KUKA KRL program: Rack_Azul_Dejar.src, Rack_Azul_Dejar.dat

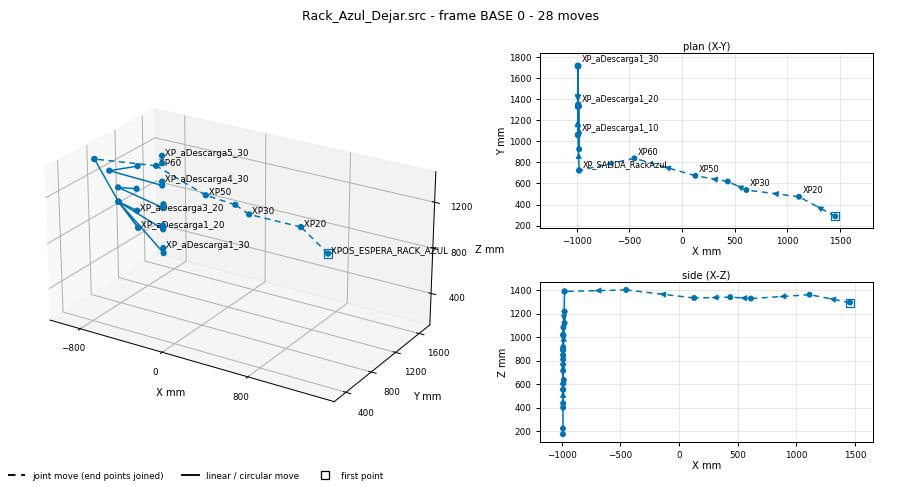
[picture p0: tool path of Rack_Azul_Dejar.src in frame BASE 0, 28 of 41 moves have a stored position in this frame; points joined in program order, loops and branches not executed]
--- Rack_Azul_Dejar.src ---
&ACCESS RVO1
&REL 3149
&COMMENT DEJAR BAT EN RACK AZUL
&PARAM EDITMASK = *
&PARAM TEMPLATE = C:\KRC\Roboter\Template\vorgabe
&PARAM DISKPATH = KRC:\R1\Program\MAFELEC
DEF Rack_Azul_Dejar( )
;FOLD INI;%{PE}
  ;FOLD BASISTECH INI
    GLOBAL INTERRUPT DECL 3 WHEN $STOPMESS==TRUE DO IR_STOPM ( )
    INTERRUPT ON 3
    BAS (#INITMOV,0 )
  ;ENDFOLD (BASISTECH INI)
;FOLD SPOTTECH INI
USERSPOT(#INIT)
;ENDFOLD (SPOTTECH INI)
;FOLD GRIPPERTECH INI
USER_GRP(0,DUMMY,DUMMY,GDEFAULT)
;ENDFOLD (GRIPPERTECH INI)
;FOLD USER INI
INTERRUPT DECL 26 WHEN I_121R1S102 OR I_121R1S202 DO PARO_RAPIDO ()
INTERRUPT DECL 27 WHEN I_121R1S302 OR I_121R1S402 DO PARO_RAPIDO ()
    ;Make your modifications here
O_TYPE_INFO=0
SELECT_T1=FALSE

  ;ENDFOLD (USER INI)
;ENDFOLD (INI)
;################################################
; PROYECTO: MAFELEC PLANTA DE BATERIAS
; ROBOT: 121_R1
; PROGRAMA: DESCARGA DE BATERIA EN RACK AZUL
; CREADO POR: Mike Tyson(zaisor robotics)
; FECHA: 23-NOVIEMBRE-2022
; MODIFICADO POR:
; FECHA MODIFICACION: 17-ENERO-2023
;################################################

; FOLD CARGA VALORES DE POSICION
IF FRAME_POS.A < 180.0 THEN
FRAME_POS.A = FRAME_POS.A + 360
ENDIF
IF FRAME_POS.B < 180.0 THEN
FRAME_POS.B = FRAME_POS.B + 360
ENDIF
IF FRAME_POS.C < 180.0 THEN
FRAME_POS.C = FRAME_POS.C + 360
ENDIF

IF FRAME_POS.A > 180.0 THEN
FRAME_POS.A = FRAME_POS.A - 360
ENDIF
IF FRAME_POS.B > 180.0 THEN
FRAME_POS.B = FRAME_POS.B - 360
ENDIF
IF FRAME_POS.C > 180.0 THEN
FRAME_POS.C = FRAME_POS.C - 360
ENDIF

XP_DEJAR_AZUL=FRAME_POS
XP_DEJAR_AZUL.z=FRAME_POS.z+3
XP_DROP_1=XP_DEJAR_AZUL
XP_DROP_2=XP_DEJAR_AZUL
XP_DROP_3=XP_DEJAR_AZUL
XP_DROP_4=XP_DEJAR_AZUL
XP_DROP_5=XP_DEJAR_AZUL

XP_DROP_1.z=XP_DROP_1.z + 80
XP_DROP_2.z=XP_DROP_2.z + 80
XP_DROP_3.z=XP_DROP_3.z + 80
XP_DROP_4.z=XP_DROP_4.z + 80
XP_DROP_5.z=XP_DROP_5.z + 80
;ENDFOLD

;FOLD PTP POS_ESPERA_RACK_AZUL Vel=100 % H Tool[11]:T_Gripper1_Carga Base[0];%{PE}%R 8.3.48,%MKUKATPBASIS,%CMOVE,%VPTP,%P 1:PTP, 2:POS_ESPERA_RACK_AZUL, 3:, 5:100, 7:H
$BWDSTART=FALSE
PDAT_ACT=PH
FDAT_ACT=FPOS_ESPERA_RACK_AZUL
BAS(#PTP_PARAMS,100)
PTP XPOS_ESPERA_RACK_AZUL
;ENDFOLD

;ESPERA AREA 2
WAIT FOR I_ARDY_2
O_AREL_2=FALSE

Empujador(1,"R",TRUE)
Empujador(2,"R",TRUE)

;FOLD PTP P20 CONT Vel=100 % M Tool[11]:T_Gripper1_Carga Base[0];%{PE}%R 8.3.48,%MKUKATPBASIS,%CMOVE,%VPTP,%P 1:PTP, 2:P20, 3:C_DIS, 5:100, 7:M
$BWDSTART=FALSE
PDAT_ACT=PM
FDAT_ACT=FP20
BAS(#PTP_PARAMS,100)
PTP XP20 C_DIS
;ENDFOLD

;FOLD PTP P30 CONT Vel=100 % M Tool[11]:T_Gripper1_Carga Base[0];%{PE}%R 8.3.48,%MKUKATPBASIS,%CMOVE,%VPTP,%P 1:PTP, 2:P30, 3:C_DIS, 5:100, 7:M
$BWDSTART=FALSE
PDAT_ACT=PM
FDAT_ACT=FP30
BAS(#PTP_PARAMS,100)
PTP XP30 C_DIS
;ENDFOLD
;FOLD PTP P40 CONT Vel=100 % M Tool[11]:T_Gripper1_Carga Base[0];%{PE}%R 8.3.48,%MKUKATPBASIS,%CMOVE,%VPTP,%P 1:PTP, 2:P40, 3:C_DIS, 5:100, 7:M
$BWDSTART=FALSE
PDAT_ACT=PM
FDAT_ACT=FP40
BAS(#PTP_PARAMS,100)
PTP XP40 C_DIS
;ENDFOLD
;FOLD PTP P50 CONT Vel=100 % M Tool[11]:T_Gripper1_Carga Base[0];%{PE}%R 8.3.48,%MKUKATPBASIS,%CMOVE,%VPTP,%P 1:PTP, 2:P50, 3:C_DIS, 5:100, 7:M
$BWDSTART=FALSE
PDAT_ACT=PM
FDAT_ACT=FP50
BAS(#PTP_PARAMS,100)
PTP XP50 C_DIS
;ENDFOLD
;FOLD PTP P60 CONT Vel=100 % L Tool[11]:T_Gripper1_Carga Base[0];%{PE}%R 8.3.48,%MKUKATPBASIS,%CMOVE,%VPTP,%P 1:PTP, 2:P60, 3:C_DIS, 5:100, 7:L
$BWDSTART=FALSE
PDAT_ACT=PL
FDAT_ACT=FP60
BAS(#PTP_PARAMS,100)
PTP XP60 C_DIS
;ENDFOLD

; POSICION DE ESPERA A DEJAR BATERIA EN RACK AZUL
;FOLD PTP P_Espera_Dejar_Rack_A Vel=50 % L Tool[11]:T_Gripper1_Carga Base[0];%{PE}%R 8.3.48,%MKUKATPBASIS,%CMOVE,%VPTP,%P 1:PTP, 2:P_Espera_Dejar_Rack_A, 3:, 5:50, 7:L
$BWDSTART=FALSE
PDAT_ACT=PL
FDAT_ACT=FP_Espera_Dejar_Rack_A
BAS(#PTP_PARAMS,50)
PTP XP_Espera_Dejar_Rack_A
;ENDFOLD

; FOLD ACTIVA VIGILANCIA SOBREPASO
;INTERRUPT ON 26
;INTERRUPT ON 27
;ENDFOLD

;CONTROL DE AUSENCIA DE PIEZA EN GRIPPER
IF (I_SIMULACION==FALSE) THEN
IF NOT I_121R1S1000 THEN
HALT
ENDIF
ENDIF

;FOLD CONTROL APERTURA GRIPPER
IF (I_121R1S131A==FALSE) OR (I_121R1S132A==FALSE) OR (I_121R1S133A==FALSE) OR (I_121R1S134A==FALSE) THEN
HALT
ENDIF
;ENDFOLD

IF PGNO==21 THEN
O_TYPE_RQ=TRUE
WAIT FOR (I_TYPE_INFO>20) AND (I_TYPE_INFO<26)
RA_Bandeja_Nr=I_TYPE_INFO
O_TYPE_RQ=FALSE
ENDIF

WAIT FOR (RA_Bandeja_Nr>20) AND (RA_Bandeja_Nr<26)

SWITCH RA_Bandeja_Nr ;

CASE 21
; MOVIMIENTOS HACIA BANDEJA 1
O_TYPE_INFO=21

WAIT FOR I_Rack2_S1==TRUE
;FOLD LIN P_aDescarga1_10 CONT Vel=0.5 m/s L Tool[11]:T_Gripper1_Carga Base[0];%{PE}%R 8.3.48,%MKUKATPBASIS,%CMOVE,%VLIN,%P 1:LIN, 2:P_aDescarga1_10, 3:C_DIS C_DIS, 5:0.5, 7:L
$BWDSTART=FALSE
LDAT_ACT=LL
FDAT_ACT=FP_aDescarga1_10
BAS(#CP_PARAMS,0.5)
LIN XP_aDescarga1_10 C_DIS C_DIS
;ENDFOLD
;FOLD LIN P_aDescarga1_20 CONT Vel=0.5 m/s L Tool[11]:T_Gripper1_Carga Base[0];%{PE}%R 8.3.48,%MKUKATPBASIS,%CMOVE,%VLIN,%P 1:LIN, 2:P_aDescarga1_20, 3:C_DIS C_DIS, 5:0.5, 7:L
$BWDSTART=FALSE
LDAT_ACT=LL
FDAT_ACT=FP_aDescarga1_20
BAS(#CP_PARAMS,0.5)
LIN XP_aDescarga1_20 C_DIS C_DIS
;ENDFOLD

IF (O_INPICKER_OK==TRUE) AND (O_INPICKER_NOK==FALSE) THEN
; #### MOVIMIENTOS A DESCARGA CONTROLADOS POR ####
; #### LA CAMARA DE VISION                    ####

;FOLD LIN P_DROP_1 Vel=0.3 m/s L Tool[11]:T_Gripper1_Carga Base[0];%{PE}%R 8.3.48,%MKUKATPBASIS,%CMOVE,%VLIN,%P 1:LIN, 2:P_DROP_1, 3:, 5:0.3, 7:L
$BWDSTART=FALSE
LDAT_ACT=LL
FDAT_ACT=FP_DROP_1
BAS(#CP_PARAMS,0.3)
LIN XP_DROP_1
;ENDFOLD
;FOLD LIN P_DEJAR_AZUL Vel=0.1 m/s L Tool[11]:T_Gripper1_Carga Base[0];%{PE}%R 8.3.48,%MKUKATPBASIS,%CMOVE,%VLIN,%P 1:LIN, 2:P_DEJAR_AZUL, 3:, 5:0.1, 7:L
$BWDSTART=FALSE
LDAT_ACT=LL
FDAT_ACT=FP_DEJAR_AZUL
BAS(#CP_PARAMS,0.1)
LIN XP_DEJAR_AZUL
;ENDFOLD

ELSE

; #### MOVIMIENTOS A DESCARGA CONTROLADOS POR ####
; #### EL OPERARIO                            ####
;FOLD ESPERA LLAVE SELECTORA EN MODO T1
WAIT FOR $T1
SELECT_T1=TRUE
;ENDFOLD
;FOLD LIN P_aDescarga1_30 CONT Vel=0.2 m/s L Tool[11]:T_Gripper1_Carga Base[0];%{PE}%R 8.3.48,%MKUKATPBASIS,%CMOVE,%VLIN,%P 1:LIN, 2:P_aDescarga1_30, 3:C_DIS C_DIS, 5:0.2, 7:L
$BWDSTART=FALSE
LDAT_ACT=LL
FDAT_ACT=FP_aDescarga1_30
BAS(#CP_PARAMS,0.2)
LIN XP_aDescarga1_30 C_DIS C_DIS
;ENDFOLD

;POSICION DE DESCARGA 1
;CUIDADO CON EL LINEAL NO EJECUTARLO HASTA EL FINAL
;POSIBILIDAD DE COLISION
;EN ESTE PUNTO LLEVAR EL ROBOT HASTA LA DESCARGA DE BANDEJA
;UNA VEZ TENEMOS EL ROBOT YA EN LA POSICION DE DEJADA TENEMOS
;QUE ACTIVAR LAS SALIDAS DE LAS CLAMPAS PARA DEJAR LA BATERIA
;SALIDA 246 O_121R1Y13A PINES BLOQUEO ADELANTE ESTARA EN 1 PONERLA A 0
;SEGUIDAMENTE LA SALIDA 245 O_121R1Y13B PINES BLOQUEO ATRAS ESTARA A 0 PONERLA A 1
;AL ABRIR LOS PINES DE LAS CLAMPAS EL SIGUIENTE PASO ES SELECCIONAR LA LINEA
;ENDIF Y CONTINUAR PROGRAMA
;FOLD LIN Rack_Azul_Pos1 Vel=0.2 m/s L Tool[11]:T_Gripper1_Carga Base[0];%{PE}%R 8.3.48,%MKUKATPBASIS,%CMOVE,%VLIN,%P 1:LIN, 2:Rack_Azul_Pos1, 3:, 5:0.2, 7:L
$BWDSTART=FALSE
LDAT_ACT=LL
FDAT_ACT=FRack_Azul_Pos1
BAS(#CP_PARAMS,0.2)
LIN XRack_Azul_Pos1
;ENDFOLD
ENDIF

CASE 22
O_TYPE_INFO=22
; MOVIMIENTOS HACIA BANDEJA 2
WAIT FOR I_Rack2_S2==TRUE
;FOLD LIN P_aDescarga2_10 CONT Vel=0.5 m/s L Tool[11]:T_Gripper1_Carga Base[0];%{PE}%R 8.3.48,%MKUKATPBASIS,%CMOVE,%VLIN,%P 1:LIN, 2:P_aDescarga2_10, 3:C_DIS C_DIS, 5:0.5, 7:L
$BWDSTART=FALSE
LDAT_ACT=LL
FDAT_ACT=FP_aDescarga2_10
BAS(#CP_PARAMS,0.5)
LIN XP_aDescarga2_10 C_DIS C_DIS
;ENDFOLD
;FOLD LIN P_aDescarga2_20 CONT Vel=0.5 m/s L Tool[11]:T_Gripper1_Carga Base[0];%{PE}%R 8.3.48,%MKUKATPBASIS,%CMOVE,%VLIN,%P 1:LIN, 2:P_aDescarga2_20, 3:C_DIS C_DIS, 5:0.5, 7:L
$BWDSTART=FALSE
LDAT_ACT=LL
FDAT_ACT=FP_aDescarga2_20
BAS(#CP_PARAMS,0.5)
LIN XP_aDescarga2_20 C_DIS C_DIS
;ENDFOLD

IF (O_INPICKER_OK==TRUE) AND (O_INPICKER_NOK==FALSE) AND (O_LIMITS_OK==TRUE) AND (O_LIMITS_NOK==FALSE) THEN
; #### MOVIMIENTOS A DESCARGA CONTROLADOS POR ####
; #### LA CAMARA DE VISION                    ####

;FOLD LIN P_DROP_2 Vel=0.3 m/s L Tool[11]:T_Gripper1_Carga Base[0];%{PE}%R 8.3.48,%MKUKATPBASIS,%CMOVE,%VLIN,%P 1:LIN, 2:P_DROP_2, 3:, 5:0.3, 7:L
$BWDSTART=FALSE
LDAT_ACT=LL
FDAT_ACT=FP_DROP_2
BAS(#CP_PARAMS,0.3)
LIN XP_DROP_2
;ENDFOLD
;FOLD LIN P_DEJAR_AZUL Vel=0.1 m/s L Tool[11]:T_Gripper1_Carga Base[0];%{PE}%R 8.3.48,%MKUKATPBASIS,%CMOVE,%VLIN,%P 1:LIN, 2:P_DEJAR_AZUL, 3:, 5:0.1, 7:L
$BWDSTART=FALSE
LDAT_ACT=LL
FDAT_ACT=FP_DEJAR_AZUL
BAS(#CP_PARAMS,0.1)
LIN XP_DEJAR_AZUL
;ENDFOLD

ELSE
; #### MOVIMIENTOS A DESCARGA CONTROLADOS POR ####
; #### EL OPERARIO                            ####
;FOLD ESPERA LLAVE SELECTORA EN MODO T1
WAIT FOR $T1
SELECT_T1=TRUE
;ENDFOLD
;FOLD LIN P_aDescarga2_30 CONT Vel=0.2 m/s L Tool[11]:T_Gripper1_Carga Base[0];%{PE}%R 8.3.48,%MKUKATPBASIS,%CMOVE,%VLIN,%P 1:LIN, 2:P_aDescarga2_30, 3:C_DIS C_DIS, 5:0.2, 7:L
$BWDSTART=FALSE
LDAT_ACT=LL
FDAT_ACT=FP_aDescarga2_30
BAS(#CP_PARAMS,0.2)
LIN XP_aDescarga2_30 C_DIS C_DIS
;ENDFOLD

;POSICION DE DESCARGA 2
;CUIDADO CON EL LINEAL NO EJECUTARLO HASTA EL FINAL
;POSIBILIDAD DE COLISION
;EN ESTE PUNTO LLEVAR EL ROBOT HASTA LA DESCARGA DE BANDEJA
;UNA VEZ TENEMOS EL ROBOT YA EN LA POSICION DE DEJADA TENEMOS
;QUE ACTIVAR LAS SALIDAS DE LAS CLAMPAS PARA DEJAR LA BATERIA
;SALIDA 246 O_121R1Y13A PINES BLOQUEO ADELANTE ESTARA EN 1 PONERLA A 0
;SEGUIDAMENTE LA SALIDA 245 O_121R1Y13B PINES BLOQUEO ATRAS ESTARA A 0 PONERLA A 1
;AL ABRIR LOS PINES DE LAS CLAMPAS EL SIGUIENTE PASO ES SELECCIONAR LA LINEA
;ENDIF Y CONTINUAR PROGRAMA
;FOLD LIN Rack_Azul_Pos2 Vel=0.2 m/s L Tool[11]:T_Gripper1_Carga Base[0];%{PE}%R 8.3.48,%MKUKATPBASIS,%CMOVE,%VLIN,%P 1:LIN, 2:Rack_Azul_Pos2, 3:, 5:0.2, 7:L
$BWDSTART=FALSE
LDAT_ACT=LL
FDAT_ACT=FRack_Azul_Pos2
BAS(#CP_PARAMS,0.2)
LIN XRack_Azul_Pos2
;ENDFOLD
ENDIF

CASE 23
; MOVIMIENTOS HACIA BANDEJA 3
O_TYPE_INFO=23
WAIT FOR I_Rack2_S3==TRUE
;FOLD LIN P_aDescarga3_10 CONT Vel=0.5 m/s L Tool[11]:T_Gripper1_Carga Base[0];%{PE}%R 8.3.48,%MKUKATPBASIS,%CMOVE,%VLIN,%P 1:LIN, 2:P_aDescarga3_10, 3:C_DIS C_DIS, 5:0.5, 7:L
$BWDSTART=FALSE
LDAT_ACT=LL
FDAT_ACT=FP_aDescarga3_10
BAS(#CP_PARAMS,0.5)
LIN XP_aDescarga3_10 C_DIS C_DIS
;ENDFOLD
;FOLD LIN P_aDescarga3_20 CONT Vel=0.5 m/s L Tool[11]:T_Gripper1_Carga Base[0];%{PE}%R 8.3.48,%MKUKATPBASIS,%CMOVE,%VLIN,%P 1:LIN, 2:P_aDescarga3_20, 3:C_DIS C_DIS, 5:0.5, 7:L
$BWDSTART=FALSE
LDAT_ACT=LL
FDAT_ACT=FP_aDescarga3_20
BAS(#CP_PARAMS,0.5)
LIN XP_aDescarga3_20 C_DIS C_DIS
;ENDFOLD


IF (O_INPICKER_OK==TRUE) AND (O_INPICKER_NOK==FALSE) AND (O_LIMITS_OK==TRUE) AND (O_LIMITS_NOK==FALSE) THEN
; #### MOVIMIENTOS A DESCARGA CONTROLADOS POR ####
; #### LA CAMARA DE VISION                    ####

;FOLD LIN P_DROP_3 Vel=0.3 m/s L Tool[11]:T_Gripper1_Carga Base[0];%{PE}%R 8.3.48,%MKUKATPBASIS,%CMOVE,%VLIN,%P 1:LIN, 2:P_DROP_3, 3:, 5:0.3, 7:L
$BWDSTART=FALSE
LDAT_ACT=LL
FDAT_ACT=FP_DROP_3
BAS(#CP_PARAMS,0.3)
LIN XP_DROP_3
;ENDFOLD
;FOLD LIN P_DEJAR_AZUL Vel=0.1 m/s L Tool[11]:T_Gripper1_Carga Base[0];%{PE}%R 8.3.48,%MKUKATPBASIS,%CMOVE,%VLIN,%P 1:LIN, 2:P_DEJAR_AZUL, 3:, 5:0.1, 7:L
$BWDSTART=FALSE
LDAT_ACT=LL
FDAT_ACT=FP_DEJAR_AZUL
BAS(#CP_PARAMS,0.1)
LIN XP_DEJAR_AZUL
;ENDFOLD

ELSE
; #### MOVIMIENTOS A DESCARGA CONTROLADOS POR ####
; #### EL OPERARIO                            ####
;FOLD ESPERA LLAVE SELECTORA EN MODO T1
WAIT FOR $T1
SELECT_T1=TRUE
;ENDFOLD
;FOLD LIN P_aDescarga3_30 CONT Vel=0.2 m/s L Tool[11]:T_Gripper1_Carga Base[0];%{PE}%R 8.3.48,%MKUKATPBASIS,%CMOVE,%VLIN,%P 1:LIN, 2:P_aDescarga3_30, 3:C_DIS C_DIS, 5:0.2, 7:L
$BWDSTART=FALSE
LDAT_ACT=LL
FDAT_ACT=FP_aDescarga3_30
BAS(#CP_PARAMS,0.2)
LIN XP_aDescarga3_30 C_DIS C_DIS
;ENDFOLD

;POSICION DE DESCARGA 3
;CUIDADO CON EL LINEAL NO EJECUTARLO HASTA EL FINAL
;POSIBILIDAD DE COLISION
;EN ESTE PUNTO LLEVAR EL ROBOT HASTA LA DESCARGA DE BANDEJA
;UNA VEZ TENEMOS EL ROBOT YA EN LA POSICION DE DEJADA TENEMOS
;QUE ACTIVAR LAS SALIDAS DE LAS CLAMPAS PARA DEJAR LA BATERIA
;SALIDA 246 O_121R1Y13A PINES BLOQUEO ADELANTE ESTARA EN 1 PONERLA A 0
;SEGUIDAMENTE LA SALIDA 245 O_121R1Y13B PINES BLOQUEO ATRAS ESTARA A 0 PONERLA A 1
;AL ABRIR LOS PINES DE LAS CLAMPAS EL SIGUIENTE PASO ES SELECCIONAR LA LINEA
;ENDIF Y CONTINUAR PROGRAMA
;FOLD LIN Rack_Azul_Pos3 Vel=0.2 m/s L Tool[11]:T_Gripper1_Carga Base[0];%{PE}%R 8.3.48,%MKUKATPBASIS,%CMOVE,%VLIN,%P 1:LIN, 2:Rack_Azul_Pos3, 3:, 5:0.2, 7:L
$BWDSTART=FALSE
LDAT_ACT=LL
FDAT_ACT=FRack_Azul_Pos3
BAS(#CP_PARAMS,0.2)
LIN XRack_Azul_Pos3
;ENDFOLD
ENDIF

CASE 24
; MOVIMIENTOS HACIA BANDEJA4
O_TYPE_INFO=24
WAIT FOR I_Rack2_S4==TRUE
;FOLD LIN P_aDescarga4_10 CONT Vel=0.5 m/s L Tool[11]:T_Gripper1_Carga Base[0];%{PE}%R 8.3.48,%MKUKATPBASIS,%CMOVE,%VLIN,%P 1:LIN, 2:P_aDescarga4_10, 3:C_DIS C_DIS, 5:0.5, 7:L
$BWDSTART=FALSE
LDAT_ACT=LL
FDAT_ACT=FP_aDescarga4_10
BAS(#CP_PARAMS,0.5)
LIN XP_aDescarga4_10 C_DIS C_DIS
;ENDFOLD
;FOLD LIN P_aDescarga4_20 CONT Vel=0.5 m/s L Tool[11]:T_Gripper1_Carga Base[0];%{PE}%R 8.3.48,%MKUKATPBASIS,%CMOVE,%VLIN,%P 1:LIN, 2:P_aDescarga4_20, 3:C_DIS C_DIS, 5:0.5, 7:L
$BWDSTART=FALSE
LDAT_ACT=LL
FDAT_ACT=FP_aDescarga4_20
BAS(#CP_PARAMS,0.5)
LIN XP_aDescarga4_20 C_DIS C_DIS
;ENDFOLD

IF (O_INPICKER_OK==TRUE) AND (O_INPICKER_NOK==FALSE) AND (O_LIMITS_OK==TRUE) AND (O_LIMITS_NOK==FALSE) THEN
; #### MOVIMIENTOS A DESCARGA CONTROLADOS POR ####
; #### LA CAMARA DE VISION                    ####

;FOLD LIN P_DROP_4 Vel=0.3 m/s L Tool[11]:T_Gripper1_Carga Base[0];%{PE}%R 8.3.48,%MKUKATPBASIS,%CMOVE,%VLIN,%P 1:LIN, 2:P_DROP_4, 3:, 5:0.3, 7:L
$BWDSTART=FALSE
LDAT_ACT=LL
FDAT_ACT=FP_DROP_4
BAS(#CP_PARAMS,0.3)
LIN XP_DROP_4
;ENDFOLD
;FOLD LIN P_DEJAR_AZUL Vel=0.1 m/s L Tool[11]:T_Gripper1_Carga Base[0];%{PE}%R 8.3.48,%MKUKATPBASIS,%CMOVE,%VLIN,%P 1:LIN, 2:P_DEJAR_AZUL, 3:, 5:0.1, 7:L
$BWDSTART=FALSE
LDAT_ACT=LL
FDAT_ACT=FP_DEJAR_AZUL
BAS(#CP_PARAMS,0.1)
LIN XP_DEJAR_AZUL
;ENDFOLD

ELSE
; #### MOVIMIENTOS A DESCARGA CONTROLADOS POR ####
; #### EL OPERARIO                            ####
;FOLD ESPERA LLAVE SELECTORA EN MODO T1
WAIT FOR $T1
SELECT_T1=TRUE
;ENDFOLD
;FOLD LIN P_aDescarga4_30 CONT Vel=0.2 m/s L Tool[11]:T_Gripper1_Carga Base[0];%{PE}%R 8.3.48,%MKUKATPBASIS,%CMOVE,%VLIN,%P 1:LIN, 2:P_aDescarga4_30, 3:C_DIS C_DIS, 5:0.2, 7:L
$BWDSTART=FALSE
LDAT_ACT=LL
FDAT_ACT=FP_aDescarga4_30
BAS(#CP_PARAMS,0.2)
LIN XP_aDescarga4_30 C_DIS C_DIS
;ENDFOLD

;POSICION DE DESCARGA 4
;CUIDADO CON EL LINEAL NO EJECUTARLO HASTA EL FINAL
;POSIBILIDAD DE COLISION
;EN ESTE PUNTO LLEVAR EL ROBOT HASTA LA DESCARGA DE BANDEJA
;UNA VEZ TENEMOS EL ROBOT YA EN LA POSICION DE DEJADA TENEMOS
;QUE ACTIVAR LAS SALIDAS DE LAS CLAMPAS PARA DEJAR LA BATERIA
;SALIDA 246 O_121R1Y13A PINES BLOQUEO ADELANTE ESTARA EN 1 PONERLA A 0
;SEGUIDAMENTE LA SALIDA 245 O_121R1Y13B PINES BLOQUEO ATRAS ESTARA A 0 PONERLA A 1
;AL ABRIR LOS PINES DE LAS CLAMPAS EL SIGUIENTE PASO ES SELECCIONAR LA LINEA
;ENDIF Y CONTINUAR PROGRAMA
;FOLD LIN Rack_Azul_Pos4 Vel=0.2 m/s L Tool[11]:T_Gripper1_Carga Base[0];%{PE}%R 8.3.48,%MKUKATPBASIS,%CMOVE,%VLIN,%P 1:LIN, 2:Rack_Azul_Pos4, 3:, 5:0.2, 7:L
$BWDSTART=FALSE
LDAT_ACT=LL
FDAT_ACT=FRack_Azul_Pos4
BAS(#CP_PARAMS,0.2)
LIN XRack_Azul_Pos4
;ENDFOLD
ENDIF

CASE 25
; MOVIMIENTOS HACIA BANDEJA 5
O_TYPE_INFO=25
WAIT FOR I_Rack2_S5==TRUE
;FOLD LIN P_aDescarga5_10 CONT Vel=0.5 m/s L Tool[11]:T_Gripper1_Carga Base[0];%{PE}%R 8.3.48,%MKUKATPBASIS,%CMOVE,%VLIN,%P 1:LIN, 2:P_aDescarga5_10, 3:C_DIS C_DIS, 5:0.5, 7:L
$BWDSTART=FALSE
LDAT_ACT=LL
FDAT_ACT=FP_aDescarga5_10
BAS(#CP_PARAMS,0.5)
LIN XP_aDescarga5_10 C_DIS C_DIS
;ENDFOLD
;FOLD LIN P_aDescarga5_20 CONT Vel=0.5 m/s L Tool[11]:T_Gripper1_Carga Base[0];%{PE}%R 8.3.48,%MKUKATPBASIS,%CMOVE,%VLIN,%P 1:LIN, 2:P_aDescarga5_20, 3:C_DIS C_DIS, 5:0.5, 7:L
$BWDSTART=FALSE
LDAT_ACT=LL
FDAT_ACT=FP_aDescarga5_20
BAS(#CP_PARAMS,0.5)
LIN XP_aDescarga5_20 C_DIS C_DIS
;ENDFOLD

IF (O_INPICKER_OK==TRUE) AND (O_INPICKER_NOK==FALSE) AND (O_LIMITS_OK==TRUE) AND (O_LIMITS_NOK==FALSE) THEN

; #### MOVIMIENTOS A DESCARGA CONTROLADOS POR ####
; #### LA CAMARA DE VISION                    ####

;FOLD LIN P_DROP_5 Vel=0.3 m/s L Tool[11]:T_Gripper1_Carga Base[0];%{PE}%R 8.3.48,%MKUKATPBASIS,%CMOVE,%VLIN,%P 1:LIN, 2:P_DROP_5, 3:, 5:0.3, 7:L
$BWDSTART=FALSE
LDAT_ACT=LL
FDAT_ACT=FP_DROP_5
BAS(#CP_PARAMS,0.3)
LIN XP_DROP_5
;ENDFOLD
;FOLD LIN P_DEJAR_AZUL Vel=0.1 m/s L Tool[11]:T_Gripper1_Carga Base[0];%{PE}%R 8.3.48,%MKUKATPBASIS,%CMOVE,%VLIN,%P 1:LIN, 2:P_DEJAR_AZUL, 3:, 5:0.1, 7:L
$BWDSTART=FALSE
LDAT_ACT=LL
FDAT_ACT=FP_DEJAR_AZUL
BAS(#CP_PARAMS,0.1)
LIN XP_DEJAR_AZUL
;ENDFOLD

ELSE
; #### MOVIMIENTOS A DESCARGA CONTROLADOS POR ####
; #### EL OPERARIO                            ####
;FOLD ESPERA LLAVE SELECTORA EN MODO T1
WAIT FOR $T1
SELECT_T1=TRUE
;ENDFOLD
;FOLD LIN P_aDescarga5_30 CONT Vel=0.2 m/s L Tool[11]:T_Gripper1_Carga Base[0];%{PE}%R 8.3.48,%MKUKATPBASIS,%CMOVE,%VLIN,%P 1:LIN, 2:P_aDescarga5_30, 3:C_DIS C_DIS, 5:0.2, 7:L
$BWDSTART=FALSE
LDAT_ACT=LL
FDAT_ACT=FP_aDescarga5_30
BAS(#CP_PARAMS,0.2)
LIN XP_aDescarga5_30 C_DIS C_DIS
;ENDFOLD

;POSICION DE DESCARGA 5
;CUIDADO CON EL LINEAL NO EJECUTARLO HASTA EL FINAL
;POSIBILIDAD DE COLISION
;EN ESTE PUNTO LLEVAR EL ROBOT HASTA LA DESCARGA DE BANDEJA
;UNA VEZ TENEMOS EL ROBOT YA EN LA POSICION DE DEJADA TENEMOS
;QUE ACTIVAR LAS SALIDAS DE LAS CLAMPAS PARA DEJAR LA BATERIA
;SALIDA 246 O_121R1Y13A PINES BLOQUEO ADELANTE ESTARA EN 1 PONERLA A 0
;SEGUIDAMENTE LA SALIDA 245 O_121R1Y13B PINES BLOQUEO ATRAS ESTARA A 0 PONERLA A 1
;AL ABRIR LOS PINES DE LAS CLAMPAS EL SIGUIENTE PASO ES SELECCIONAR LA LINEA
;ENDIF Y CONTINUAR PROGRAMA
;FOLD LIN Rack_Azul_Pos5 Vel=0.2 m/s L Tool[11]:T_Gripper1_Carga Base[0];%{PE}%R 8.3.48,%MKUKATPBASIS,%CMOVE,%VLIN,%P 1:LIN, 2:Rack_Azul_Pos5, 3:, 5:0.2, 7:L
$BWDSTART=FALSE
LDAT_ACT=LL
FDAT_ACT=FRack_Azul_Pos5
BAS(#CP_PARAMS,0.2)
LIN XRack_Azul_Pos5
;ENDFOLD
ENDIF

DEFAULT

HALT
HALT
; #### CODIGO DE DESCARGA ERRONEO ####
HALT
BRAKE
ENDSWITCH

; FOLD MOVIMIENTOS DE SALIDA RACK AZUL
INI_DROP:
GIRO_A_P=FALSE
GIRO_A_N=FALSE
GIRO_B_P=FALSE
GIRO_B_N=FALSE
GIRO_C_P=FALSE
GIRO_C_N=FALSE
PTP $POS_ACT

IF (I_SIMULACION==FALSE) THEN

Repite=0

WHILE (I_121R1S102==TRUE) OR (I_121R1S202==TRUE) OR (I_121R1S302==TRUE) OR (I_121R1S402==TRUE)

Repite=Repite+1
LIN_REL{Z +1}
WAIT SEC 0.1

IF Repite>=3 THEN
HALT
; SUPERADO NUMERO DE REPETICIONES
HALT
ENDIF

ENDWHILE

Repite=0

WHILE (I_121R1S101==FALSE) AND (I_121R1S201==FALSE) AND (I_121R1S301==FALSE) AND (I_121R1S401==FALSE)
IF (I_121R1S102==TRUE) OR (I_121R1S202==TRUE) OR (I_121R1S302==TRUE) OR (I_121R1S402==TRUE) THEN
HALT
HALT
HALT
ENDIF
Repite=Repite+1
LIN_REL{Z -1}
WAIT SEC 0.1

IF Repite>=8 THEN
HALT
; SUPERADO NUMERO DE REPETICIONES
HALT
ENDIF

ENDWHILE

; #### CONTROL DE PRESENCIA PARA ABRIR ####
WAIT FOR (I_121R1S101==TRUE) OR (I_121R1S301==TRUE) OR (I_121R1S201==TRUE) OR (I_121R1S401==TRUE)

fin_dejar:
ENDIF

O_INPICKER_OK=FALSE
O_INPICKER_NOK=FALSE
O_LIMITS_OK=FALSE
O_LIMITS_NOK=FALSE
O_LIMIT_X=FALSE
O_LIMIT_Y=FALSE
O_LIMIT_Z=FALSE
O_LIMIT_A=FALSE
O_LIMIT_B=FALSE
O_LIMIT_C=FALSE

PTP $POS_ACT
Pines("R")

PTP $POS_ACT
WAIT FOR $EXT; CAMBIAR LA LLAVE A MODO EXT

LIN_REL{Z +80}
O_JRDY_6 = TRUE
BAS(#CP_PARAMS,1.5)

; #### CONTROL DE AUSENCIA DE BATERIA ####
WAIT FOR NOT I_121R1S1000

LIN_REL{Y -300,Z +100} C_DIS
LIN_REL{Y -400,Z +350}
; ENDFOLD
; FOLD FIN VIGILANCIA SOBREPASO
INTERRUPT OFF 26
INTERRUPT OFF 27
;ENDFOLD

;FOLD LIN P_SALIDA_RackAzul Vel=0.5 m/s M Tool[9]:T_Gripper1_Vacio Base[0];%{PE}%R 8.3.48,%MKUKATPBASIS,%CMOVE,%VLIN,%P 1:LIN, 2:P_SALIDA_RackAzul, 3:, 5:0.5, 7:M
$BWDSTART=FALSE
LDAT_ACT=LM
FDAT_ACT=FP_SALIDA_RackAzul
BAS(#CP_PARAMS,0.5)
LIN XP_SALIDA_RackAzul
;ENDFOLD



Rack_Azul_Cerrar_D()

;TRABAJO REALIZADO
O_JRDY_7 = TRUE

END
DEF Descarga_B1()
END
DEF Descarga_B2()
END
DEF Descarga_B3()
END
DEF Descarga_B4()
END
DEF Descarga_B5()
END
DEF PARO_RAPIDO ()
BRAKE F
END

--- Rack_Azul_Dejar.dat ---
&ACCESS RVO1
&REL 3149
&COMMENT DEJAR BAT EN RACK AZUL
&PARAM EDITMASK = *
&PARAM TEMPLATE = C:\KRC\Roboter\Template\vorgabe
&PARAM DISKPATH = KRC:\R1\Program\MAFELEC
DEFDAT  Rack_Azul_Dejar
;FOLD EXTERNAL DECLARATIONS;%{PE}%MKUKATPBASIS,%CEXT,%VCOMMON,%P
;FOLD GRIPPERTECH EXT
EXT  H50 (INT  :IN,INT  :IN,INT  :IN,GRP_TYP  :IN )
;ENDFOLD (GRIPPERTECH EXT)
;FOLD SPOTTECH EXT
EXT  USERSPOT (S_COMMAND  :IN,SPOT_TYPE  :IN )
;ENDFOLD (SPOTTECH EXT)
;FOLD BASISTECH EXT;%{PE}%MKUKATPBASIS,%CEXT,%VEXT,%P
EXT  BAS (BAS_COMMAND  :IN,REAL  :IN )
DECL INT SUCCESS
;ENDFOLD (BASISTECH EXT)
;FOLD USER EXT;%{E}%MKUKATPUSER,%CEXT,%VEXT,%P
;Make your modifications here

;ENDFOLD (USER EXT)
;ENDFOLD (EXTERNAL DECLARATIONS)
DECL BASIS_SUGG_T LAST_BASIS={POINT1[] "P0                      ",POINT2[] "P0                      ",CP_PARAMS[] "CPDAT0                  ",PTP_PARAMS[] "PDAT0                   ",CONT[] "                        ",CP_VEL[] "0.1                     ",PTP_VEL[] "100                     ",SYNC_PARAMS[] "SYNCDAT                 ",SPL_NAME[] "S0                      ",A_PARAMS[] "ADAT0                   "}
DECL PDAT PH={VEL 100.000,ACC 100.000,APO_DIST 100.000,APO_MODE #CDIS,GEAR_JERK 50.0000,EXAX_IGN 0}
DECL E6POS XPOS_ESPERA_DROP_RACK1={X -1005.21851,Y -395.575073,Z 1423.46069,A -87.1007538,B -0.167297319,C 179.537186,S 2,T 42,E1 0.0,E2 0.0,E3 0.0,E4 0.0,E5 0.0,E6 0.0}
DECL FDAT FPOS_ESPERA_DROP_RACK1={TOOL_NO 11,BASE_NO 0,IPO_FRAME #BASE,POINT2[] " ",TQ_STATE FALSE}
DECL E6POS XP10={X 1457.33850,Y 287.686401,Z 1296.45581,A 90.0126114,B -0.311890274,C -179.676559,S 2,T 43,E1 0.0,E2 0.0,E3 0.0,E4 0.0,E5 0.0,E6 0.0}
DECL FDAT FP10={TOOL_NO 11,BASE_NO 0,IPO_FRAME #BASE,POINT2[] " ",TQ_STATE FALSE}
DECL E6POS XP20={X 1112.71973,Y 473.868073,Z 1363.81274,A 90.0598297,B -0.560964882,C 179.735550,S 2,T 43,E1 0.0,E2 0.0,E3 0.0,E4 0.0,E5 0.0,E6 0.0}
DECL FDAT FP20={TOOL_NO 11,BASE_NO 0,IPO_FRAME #BASE,POINT2[] " ",TQ_STATE FALSE}
DECL LDAT LL={VEL 2.00000,ACC 20.0000,APO_DIST 100.000,APO_FAC 50.0000,AXIS_VEL 100.000,AXIS_ACC 100.000,ORI_TYP #VAR,CIRC_TYP #BASE,JERK_FAC 50.0000,GEAR_JERK 50.0000,EXAX_IGN 0}
DECL E6POS XRack_Verde_Pos1={X -1003.08112,Y -1697.34668,Z 167.086884,A -90.1880493,B 0.0546767898,C 179.677963,S 2,T 34,E1 0.0,E2 0.0,E3 0.0,E4 0.0,E5 0.0,E6 0.0}
DECL FDAT FRack_Verde_Pos1={TOOL_NO 11,BASE_NO 0,IPO_FRAME #BASE,POINT2[] " ",TQ_STATE FALSE}
DECL E6POS XP_aDescarga1_30={X -989.481079,Y 1716.17297,Z 223.476624,A 89.4514160,B -0.968146801,C -179.823181,S 2,T 35,E1 0.0,E2 0.0,E3 0.0,E4 0.0,E5 0.0,E6 0.0}
DECL FDAT FP_aDescarga1_30={TOOL_NO 11,BASE_NO 0,IPO_FRAME #BASE,POINT2[] " ",TQ_STATE FALSE}
DECL E6POS XP_ADESCARGA1_20={X -987.705566,Y 1341.36072,Z 554.238098,A 89.6717606,B -1.23976099,C 179.963882,S 2,T 35,E1 0.0,E2 0.0,E3 0.0,E4 0.0,E5 0.0,E6 0.0}
DECL FDAT FP_aDescarga1_20={TOOL_NO 11,BASE_NO 0,IPO_FRAME #BASE,POINT2[] " ",TQ_STATE FALSE}
DECL E6POS XP_aDescarga1_10={X -987.707214,Y 1061.81567,Z 893.140869,A 89.6717606,B -1.23976099,C 179.963882,S 2,T 35,E1 0.0,E2 0.0,E3 0.0,E4 0.0,E5 0.0,E6 0.0}
DECL FDAT FP_aDescarga1_10={TOOL_NO 11,BASE_NO 0,IPO_FRAME #BASE,POINT2[] " ",TQ_STATE FALSE}
DECL E6POS XRack_Verde_Pos2={X -995.097229,Y -1696.48059,Z 372.601105,A -90.0145721,B 0.122046471,C 179.813599,S 2,T 34,E1 0.0,E2 0.0,E3 0.0,E4 0.0,E5 0.0,E6 0.0}
DECL FDAT FRack_Verde_Pos2={TOOL_NO 11,BASE_NO 0,IPO_FRAME #BASE,POINT2[] " ",TQ_STATE FALSE}
DECL E6POS XP_aDescarga2_10={X -987.707214,Y 1061.81567,Z 893.140869,A 89.6717606,B -1.23976099,C 179.963882,S 2,T 35,E1 0.0,E2 0.0,E3 0.0,E4 0.0,E5 0.0,E6 0.0}
DECL FDAT FP_aDescarga2_10={TOOL_NO 11,BASE_NO 0,IPO_FRAME #BASE,POINT2[] " ",TQ_STATE FALSE}
DECL E6POS XP_aDescarga2_20={X -987.705566,Y 1341.36072,Z 554.238098,A 89.6717606,B -1.23976099,C 179.963882,S 2,T 35,E1 0.0,E2 0.0,E3 0.0,E4 0.0,E5 0.0,E6 0.0}
DECL FDAT FP_aDescarga2_20={TOOL_NO 11,BASE_NO 0,IPO_FRAME #BASE,POINT2[] " ",TQ_STATE FALSE}
DECL E6POS XP_aDescarga2_30={X -987.705383,Y 1715.56824,Z 437.817657,A 89.4985199,B -0.868614793,C -179.681580,S 2,T 35,E1 0.0,E2 0.0,E3 0.0,E4 0.0,E5 0.0,E6 0.0}
DECL FDAT FP_aDescarga2_30={TOOL_NO 11,BASE_NO 0,IPO_FRAME #BASE,POINT2[] " ",TQ_STATE FALSE}
DECL E6POS XRack_Verde_Pos3={X -999.936890,Y -1694.68250,Z 574.434326,A -90.0360489,B -0.174496323,C 179.625610,S 2,T 34,E1 0.0,E2 0.0,E3 0.0,E4 0.0,E5 0.0,E6 0.0}
DECL FDAT FRack_Verde_Pos3={TOOL_NO 11,BASE_NO 0,IPO_FRAME #BASE,POINT2[] " ",TQ_STATE FALSE}
DECL E6POS XP_aDescarga3_10={X -987.707214,Y 1061.81567,Z 893.140869,A 89.6717606,B -1.23976099,C 179.963882,S 2,T 35,E1 0.0,E2 0.0,E3 0.0,E4 0.0,E5 0.0,E6 0.0}
DECL FDAT FP_aDescarga3_10={TOOL_NO 11,BASE_NO 0,IPO_FRAME #BASE,POINT2[] " ",TQ_STATE FALSE}
DECL E6POS XP_aDescarga3_20={X -987.705872,Y 1330.01538,Z 715.641846,A 89.6717606,B -1.23976111,C 179.963882,S 2,T 35,E1 0.0,E2 0.0,E3 0.0,E4 0.0,E5 0.0,E6 0.0}
DECL FDAT FP_aDescarga3_20={TOOL_NO 11,BASE_NO 0,IPO_FRAME #BASE,POINT2[] " ",TQ_STATE FALSE}
DECL E6POS XP_aDescarga3_30={X -981.922424,Y 1717.76514,Z 636.524841,A 89.4239273,B -1.11692870,C -179.666199,S 2,T 35,E1 0.0,E2 0.0,E3 0.0,E4 0.0,E5 0.0,E6 0.0}
DECL FDAT FP_aDescarga3_30={TOOL_NO 11,BASE_NO 0,IPO_FRAME #BASE,POINT2[] " ",TQ_STATE FALSE}
DECL E6POS XRack_Verde_Pos4={X -995.889648,Y -1698.41321,Z 780.006104,A -89.8358231,B -0.174563199,C 179.651031,S 2,T 34,E1 0.0,E2 0.0,E3 0.0,E4 0.0,E5 0.0,E6 0.0}
DECL FDAT FRack_Verde_Pos4={TOOL_NO 11,BASE_NO 0,IPO_FRAME #BASE,POINT2[] " ",TQ_STATE FALSE}
DECL E6POS XP_aDescarga4_10={X -987.707214,Y 1061.81567,Z 1021.74384,A 89.6717606,B -1.23976099,C 179.963882,S 2,T 35,E1 0.0,E2 0.0,E3 0.0,E4 0.0,E5 0.0,E6 0.0}
DECL FDAT FP_aDescarga4_10={TOOL_NO 11,BASE_NO 0,IPO_FRAME #BASE,POINT2[] " ",TQ_STATE FALSE}
DECL E6POS XP_aDescarga4_20={X -987.707214,Y 1327.56262,Z 916.295288,A 89.6717606,B -1.23976099,C 179.963882,S 2,T 35,E1 0.0,E2 0.0,E3 0.0,E4 0.0,E5 0.0,E6 0.0}
DECL FDAT FP_aDescarga4_20={TOOL_NO 11,BASE_NO 0,IPO_FRAME #BASE,POINT2[] " ",TQ_STATE FALSE}
DECL E6POS XP_aDescarga4_30={X -987.706787,Y 1711.58740,Z 847.887,A 89.4143906,B -1.26596630,C -179.639328,S 2,T 35,E1 0.0,E2 0.0,E3 0.0,E4 0.0,E5 0.0,E6 0.0}
DECL FDAT FP_aDescarga4_30={TOOL_NO 11,BASE_NO 0,IPO_FRAME #BASE,POINT2[] " ",TQ_STATE FALSE}
DECL E6POS XRack_Verde_Pos5={X -994.762390,Y -1699.97437,Z 990.407166,A -89.9579468,B -0.567670703,C 179.413055,S 2,T 34,E1 0.0,E2 0.0,E3 0.0,E4 0.0,E5 0.0,E6 0.0}
DECL FDAT FRack_Verde_Pos5={TOOL_NO 11,BASE_NO 0,IPO_FRAME #BASE,POINT2[] " ",TQ_STATE FALSE}
DECL E6POS XP_aDescarga5_10={X -975.553406,Y 925.916504,Z 1220.19043,A 90.3743210,B -1.43819892,C -179.556488,S 2,T 35,E1 0.0,E2 0.0,E3 0.0,E4 0.0,E5 0.0,E6 0.0}
DECL FDAT FP_aDescarga5_10={TOOL_NO 11,BASE_NO 0,IPO_FRAME #BASE,POINT2[] " ",TQ_STATE FALSE}
DECL E6POS XP_aDescarga5_20={X -975.553406,Y 1332.63794,Z 1121.68311,A 90.3743210,B -1.43819892,C -179.556488,S 2,T 35,E1 0.0,E2 0.0,E3 0.0,E4 0.0,E5 0.0,E6 0.0}
DECL FDAT FP_aDescarga5_20={TOOL_NO 11,BASE_NO 0,IPO_FRAME #BASE,POINT2[] " ",TQ_STATE FALSE}
DECL E6POS XP_aDescarga5_30={X -985.364075,Y 1712.61426,Z 1084.90735,A 89.5653229,B -1.43955660,C -179.734848,S 2,T 35,E1 0.0,E2 0.0,E3 0.0,E4 0.0,E5 0.0,E6 0.0}
DECL FDAT FP_aDescarga5_30={TOOL_NO 11,BASE_NO 0,IPO_FRAME #BASE,POINT2[] " ",TQ_STATE FALSE}
DECL E6POS XP_SALIDA_RACKVERDE={X -1005.21851,Y -395.575073,Z 1423.46069,A -87.1007538,B -0.167297319,C 179.537186,S 2,T 42,E1 0.0,E2 0.0,E3 0.0,E4 0.0,E5 0.0,E6 0.0}
DECL FDAT FP_SALIDA_RackVerde={TOOL_NO 9,BASE_NO 0,IPO_FRAME #BASE,POINT2[] " ",TQ_STATE FALSE}
DECL PDAT PM={VEL 100.000,ACC 25.0000,APO_DIST 100.000,APO_MODE #CDIS,GEAR_JERK 50.0000,EXAX_IGN 0}
DECL LDAT LM={VEL 2.00000,ACC 25.0000,APO_DIST 100.000,APO_FAC 50.0000,AXIS_VEL 100.000,AXIS_ACC 100.000,ORI_TYP #VAR,CIRC_TYP #BASE,JERK_FAC 50.0000,GEAR_JERK 50.0000,EXAX_IGN 0}
DECL E6POS XP30={X 612.839355,Y 537.810791,Z 1330.94336,A 90.1527252,B -1.38403225,C 179.135300,S 2,T 43,E1 0.0,E2 0.0,E3 0.0,E4 0.0,E5 0.0,E6 0.0}
DECL FDAT FP30={TOOL_NO 11,BASE_NO 0,IPO_FRAME #BASE,POINT2[] " ",TQ_STATE FALSE}
DECL E6POS XP_DROP_1={X -983.500,Y 1705.40,Z 1076.30,A 89.7000122,B -2.00000,C -179.500}
DECL FDAT FP_DROP_1={TOOL_NO 11,BASE_NO 0,IPO_FRAME #BASE,POINT2[] " ",TQ_STATE FALSE}
DECL E6POS XP_DEJAR_AUTO={X 1606.70789,Y -354.796814,Z 1944.22656,A 1.33749425,B -32.3921471,C 179.037674,S 2,T 42,E1 0.0,E2 0.0,E3 0.0,E4 0.0,E5 0.0,E6 0.0}
DECL FDAT FP_DEJAR_AUTO={TOOL_NO 11,BASE_NO 0,IPO_FRAME #BASE,POINT2[] " ",TQ_STATE FALSE}
DECL E6POS XP_DEJAR_VERDE={X -985.800,Y -1629.40,Z 1022.60,A -87.7000122,B -2.60000610,C 179.000}
DECL FDAT FP_DEJAR_VERDE={TOOL_NO 11,BASE_NO 0,IPO_FRAME #BASE,POINT2[] " ",TQ_STATE FALSE}
DECL E6POS XP_DROP_2={X -983.500,Y 1705.40,Z 1076.30,A 89.7000122,B -2.00000,C -179.500}
DECL FDAT FP_DROP_2={TOOL_NO 11,BASE_NO 0,IPO_FRAME #BASE,POINT2[] " ",TQ_STATE FALSE}
DECL E6POS XP_DROP_3={X -983.500,Y 1705.40,Z 1076.30,A 89.7000122,B -2.00000,C -179.500}
DECL FDAT FP_DROP_3={TOOL_NO 11,BASE_NO 0,IPO_FRAME #BASE,POINT2[] " ",TQ_STATE FALSE}
DECL E6POS XP_DROP_4={X -983.500,Y 1705.40,Z 1076.30,A 89.7000122,B -2.00000,C -179.500}
DECL FDAT FP_DROP_4={TOOL_NO 11,BASE_NO 0,IPO_FRAME #BASE,POINT2[] " ",TQ_STATE FALSE}
DECL E6POS XP_DROP_5={X -983.500,Y 1705.40,Z 1076.30,A 89.7000122,B -2.00000,C -179.500}
DECL FDAT FP_DROP_5={TOOL_NO 11,BASE_NO 0,IPO_FRAME #BASE,POINT2[] " ",TQ_STATE FALSE}
DECL E6POS XP_Espera_Dejar_Rack_V={X -1005.21851,Y -395.575073,Z 1423.46069,A -87.1007538,B -0.167297319,C 179.537186,S 2,T 42,E1 0.0,E2 0.0,E3 0.0,E4 0.0,E5 0.0,E6 0.0}
DECL FDAT FP_Espera_Dejar_Rack_V={TOOL_NO 11,BASE_NO 0,IPO_FRAME #BASE,POINT2[] " ",TQ_STATE FALSE}
DECL E6POS XRack_Azul_Pos5={X -985.364075,Y 1712.61426,Z 1016.53644,A 89.5653229,B -1.43955660,C -179.734848,S 2,T 35,E1 0.0,E2 0.0,E3 0.0,E4 0.0,E5 0.0,E6 0.0}
DECL FDAT FRack_Azul_Pos5={TOOL_NO 11,BASE_NO 0,IPO_FRAME #BASE,POINT2[] " ",TQ_STATE FALSE}
DECL E6POS XP_DEJAR_AZUL={X -983.500,Y 1705.40,Z 996.300,A 89.7000122,B -2.00000,C -179.500}
DECL FDAT FP_DEJAR_AZUL={TOOL_NO 11,BASE_NO 0,IPO_FRAME #BASE,POINT2[] " ",TQ_STATE FALSE}
DECL E6POS XRack_Azul_Pos4={X -987.706787,Y 1711.58740,Z 811.998352,A 89.4143906,B -1.26596630,C -179.639328,S 2,T 35,E1 0.0,E2 0.0,E3 0.0,E4 0.0,E5 0.0,E6 0.0}
DECL FDAT FRack_Azul_Pos4={TOOL_NO 11,BASE_NO 0,IPO_FRAME #BASE,POINT2[] " ",TQ_STATE FALSE}
DECL E6POS XP_Espera_Dejar_Rack_A={X -975.553711,Y 723.196777,Z 1391.45654,A 90.3743286,B -1.43820179,C -179.556488,S 2,T 35,E1 0.0,E2 0.0,E3 0.0,E4 0.0,E5 0.0,E6 0.0}
DECL FDAT FP_Espera_Dejar_Rack_A={TOOL_NO 11,BASE_NO 0,IPO_FRAME #BASE,POINT2[] " ",TQ_STATE FALSE}
DECL E6POS XRack_Azul_Pos1={X -989.481079,Y 1720.42517,Z 174.647568,A 88.7748489,B -0.968146861,C -179.823181,S 2,T 35,E1 0.0,E2 0.0,E3 0.0,E4 0.0,E5 0.0,E6 0.0}
DECL FDAT FRack_Azul_Pos1={TOOL_NO 11,BASE_NO 0,IPO_FRAME #BASE,POINT2[] " ",TQ_STATE FALSE}
DECL E6POS XRack_Azul_Pos2={X -987.705383,Y 1715.56824,Z 401.662109,A 89.4985199,B -0.868614793,C -179.681580,S 2,T 35,E1 0.0,E2 0.0,E3 0.0,E4 0.0,E5 0.0,E6 0.0}
DECL FDAT FRack_Azul_Pos2={TOOL_NO 11,BASE_NO 0,IPO_FRAME #BASE,POINT2[] " ",TQ_STATE FALSE}
DECL E6POS XRack_Azul_Pos3={X -986.517578,Y 1712.55811,Z 605.858643,A 89.2078171,B -1.23842931,C -179.805496,S 2,T 35,E1 0.0,E2 0.0,E3 0.0,E4 0.0,E5 0.0,E6 0.0}
DECL FDAT FRack_Azul_Pos3={TOOL_NO 11,BASE_NO 0,IPO_FRAME #BASE,POINT2[] " ",TQ_STATE FALSE}
DECL E6POS XP31={X 821.592651,Y 376.528870,Z 1333.31091,A 66.5605,B -0.157429606,C -179.563858,S 2,T 43,E1 0.0,E2 0.0,E3 0.0,E4 0.0,E5 0.0,E6 0.0}
DECL FDAT FP31={TOOL_NO 11,BASE_NO 0,IPO_FRAME #BASE,POINT2[] " ",TQ_STATE FALSE}
DECL E6POS XP32={X 612.839355,Y 537.810791,Z 1330.94336,A 90.1527252,B -1.38403225,C 179.135300,S 2,T 43,E1 0.0,E2 0.0,E3 0.0,E4 0.0,E5 0.0,E6 0.0}
DECL FDAT FP32={TOOL_NO 11,BASE_NO 0,IPO_FRAME #BASE,POINT2[] " ",TQ_STATE FALSE}
DECL E6POS XP33={X 129.032791,Y 672.956726,Z 1303.56372,A 89.5664825,B -5.08658266,C -178.846436,S 2,T 43,E1 0.0,E2 0.0,E3 0.0,E4 0.0,E5 0.0,E6 0.0}
DECL FDAT FP33={TOOL_NO 11,BASE_NO 0,IPO_FRAME #BASE,POINT2[] " ",TQ_STATE FALSE}
DECL E6POS XP34={X -278.956848,Y 626.281189,Z 1304.97681,A 88.0839767,B -7.38848257,C 179.824799,S 2,T 35,E1 0.0,E2 0.0,E3 0.0,E4 0.0,E5 0.0,E6 0.0}
DECL FDAT FP34={TOOL_NO 11,BASE_NO 0,IPO_FRAME #BASE,POINT2[] " ",TQ_STATE FALSE}
DECL E6POS XPOS_ESPERA_DROP_RACK2={X -1046.34619,Y 723.196716,Z 1391.45679,A 90.3743362,B -1.43820727,C -179.556488,S 2,T 35,E1 0.0,E2 0.0,E3 0.0,E4 0.0,E5 0.0,E6 0.0}
DECL FDAT FPOS_ESPERA_DROP_RACK2={TOOL_NO 11,BASE_NO 0,IPO_FRAME #BASE,POINT2[] " ",TQ_STATE FALSE}
DECL E6POS XP40={X 436.548065,Y 618.848755,Z 1342.71338,A 82.6771469,B -2.94442844,C 179.686111,S 2,T 43,E1 0.0,E2 0.0,E3 0.0,E4 0.0,E5 0.0,E6 0.0}
DECL FDAT FP40={TOOL_NO 11,BASE_NO 0,IPO_FRAME #BASE,POINT2[] " ",TQ_STATE FALSE}
DECL E6POS XP50={X 129.032669,Y 672.956116,Z 1335.58984,A 81.6660156,B -4.88053370,C -178.159042,S 2,T 43,E1 0.0,E2 0.0,E3 0.0,E4 0.0,E5 0.0,E6 0.0}
DECL FDAT FP50={TOOL_NO 11,BASE_NO 0,IPO_FRAME #BASE,POINT2[] " ",TQ_STATE FALSE}
DECL E6POS XP60={X -450.908569,Y 839.236877,Z 1404.17847,A 86.7012482,B -2.11645436,C -178.368759,S 2,T 43,E1 0.0,E2 0.0,E3 0.0,E4 0.0,E5 0.0,E6 0.0}
DECL FDAT FP60={TOOL_NO 11,BASE_NO 0,IPO_FRAME #BASE,POINT2[] " ",TQ_STATE FALSE}
DECL E6POS XP_SALIDA_RackAzul={X -975.553711,Y 723.196777,Z 1391.45654,A 90.3743286,B -1.43820179,C -179.556488,S 2,T 35,E1 0.0,E2 0.0,E3 0.0,E4 0.0,E5 0.0,E6 0.0}
DECL FDAT FP_SALIDA_RackAzul={TOOL_NO 9,BASE_NO 0,IPO_FRAME #BASE,POINT2[] " ",TQ_STATE FALSE}
DECL E6POS XPOS_ESPERA_RACK_AZUL={X 1457.33850,Y 287.686401,Z 1296.45581,A 90.0126114,B -0.311890274,C -179.676559,S 2,T 43,E1 0.0,E2 0.0,E3 0.0,E4 0.0,E5 0.0,E6 0.0}
DECL FDAT FPOS_ESPERA_RACK_AZUL={TOOL_NO 11,BASE_NO 0,IPO_FRAME #BASE,POINT2[] " ",TQ_STATE FALSE}
DECL PDAT PL={VEL 100.000,ACC 20.0000,APO_DIST 100.000,APO_MODE #CDIS,GEAR_JERK 50.0000,EXAX_IGN 0}
ENDDAT
